FUNCTION_BLOCK NVS_AIS (* Load and Store STRING Data from NVS by Key (AIS Adapter Interface) *)
  (* Standard: 61499-2; Description: Copyright (c) 2026 Meisterschulen am Ostbahnhof This program and the accompanying materials are made available under the terms of the Eclipse Public License 2.0 which is available at https://www.eclipse.org/legal/epl-2.0/ SPDX-License-Identifier: EPL-2.0 *)
  (* Version 1.0, 2026-04-13, Franz Höpfinger, Meisterschulen am Ostbahnhof, NVStial API and implementation and/or NVStial documentation *)
  PACKAGE logiBUS::storage::esp32_nvs;
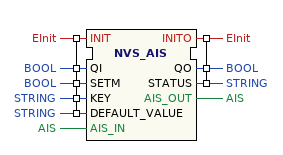
  EVENT_INPUT
    INIT : EInit WITH QI, SETM, KEY, DEFAULT_VALUE; (* Service Initialization *)
  END_EVENT
  EVENT_OUTPUT
    INITO : EInit WITH QO, STATUS; (* Initialization Confirm *)
  END_EVENT
  VAR_INPUT
    QI : BOOL; (* Event Input Qualifier *)
    SETM : BOOL; (* Enable Mirroring on SET *)
    KEY : STRING; (* Key name. *)
    DEFAULT_VALUE : STRING; (* The value to read if there is nothing in the settings.NVS *)
  END_VAR
  VAR_OUTPUT
    QO : BOOL; (* Event Output Qualifier *)
    STATUS : STRING; (* Service Status *)
  END_VAR
  SOCKETS
    AIS_IN : adapter::types::unidirectional::AIS; (* Value to store (SET) *)
  END_SOCKETS
  PLUGS
    AIS_OUT : adapter::types::unidirectional::AIS; (* Stored value output (GETO) *)
  END_PLUGS
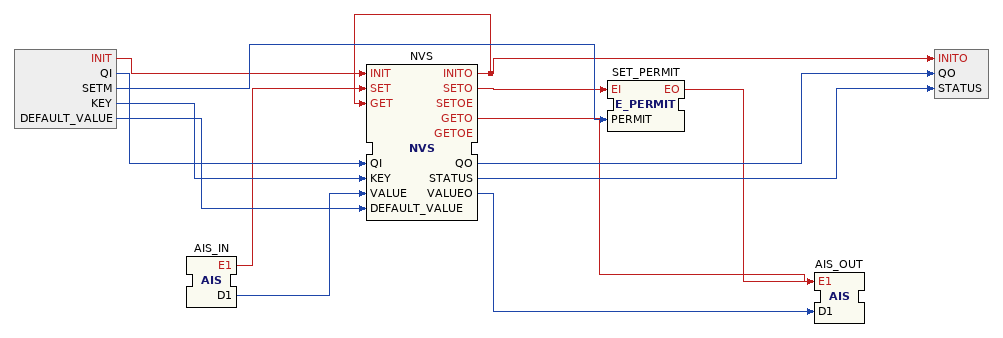
  FBS
    NVS : logiBUS::storage::esp32_nvs::NVS;
    SET_PERMIT : iec61499::events::E_PERMIT;
  END_FBS
  EVENT_CONNECTIONS
    INIT TO NVS.INIT;
    NVS.INITO TO INITO;
    NVS.INITO TO NVS.GET;
    AIS_IN.E1 TO NVS.SET;
    SET_PERMIT.EO TO AIS_OUT.E1;
    NVS.GETO TO AIS_OUT.E1;
    NVS.SETO TO SET_PERMIT.EI;
  END_CONNECTIONS
  DATA_CONNECTIONS
    QI TO NVS.QI;
    SETM TO SET_PERMIT.PERMIT;
    KEY TO NVS.KEY;
    DEFAULT_VALUE TO NVS.DEFAULT_VALUE;
    AIS_IN.D1 TO NVS.VALUE;
    NVS.VALUEO TO AIS_OUT.D1;
    NVS.QO TO QO;
    NVS.STATUS TO STATUS;
  END_CONNECTIONS
END_FUNCTION_BLOCK
